// TIA Portal V20 export
DATA_BLOCK "DB_AsiSetpoint"   // DB29
// stored: Access Published, MemoryReserve 100, Namespace LineD1
   VAR
      Line : Struct
         D1 : Struct
            DirChange : Struct
               Conveyor : Array[_.minD1.._.maxD1] of Bool;
            END_STRUCT;
            Speed : Struct
               Conveyor : Array[_.minD1.._.maxD1] of Bool;
            END_STRUCT;
         END_STRUCT;
      END_STRUCT;
   END_VAR
BEGIN
END_DATA_BLOCK
